Staubli VAL3: english.dtx

public string No = "No"
public string Yes = "Yes "
string sValProduct = "VALCLEAN"
